Staubli VAL3: extractGrid.pgx

public program extractGrid(num& x_nInput[] (dimensions=2), num x_nDimension, num x_nFrom, num x_nTo, num& x_nResult[] (dimensions=2))
  local num l_nX
  local num l_nY
  local num l_nCounter
  local num l_nStep
begin

  resize(x_nResult,1,1)
  resize(x_nResult,2,1)
  x_nResult[0,0] = -999999


  l_nCounter = 0
  if x_nDimension == 1
    resize(x_nResult,1,abs(x_nTo-x_nFrom)+1)
    resize(x_nResult,2,size(x_nInput,2))

    l_nStep = sel(x_nTo >= x_nFrom, 1, -1)

    for l_nX = x_nFrom to x_nTo step l_nStep
      for l_nY = 0 to size(x_nInput,2)-1
        x_nResult[l_nCounter, l_nY] = x_nInput[l_nX,l_nY]
      endFor
      l_nCounter = l_nCounter + 1
    endFor


  elseIf x_nDimension == 2

    resize(x_nResult,1, size(x_nInput,1))
    resize(x_nResult,2, abs(x_nTo-x_nFrom)+1)

    l_nStep = sel(x_nTo >= x_nFrom, 1, -1)

    for l_nY = x_nFrom to x_nTo step l_nStep
      for l_nX = 0 to size(x_nInput,1)-1
        x_nResult[l_nX, l_nCounter] = x_nInput[l_nX,l_nY]
      endFor
      l_nCounter = l_nCounter + 1
    endFor
  endIf

end
